SEGMENT_TYPE Ethernet (* Ethernet Segment *)
  (* Standard: 61499 ITA; Description: Copyright (c) 2008 Profactor GmbH This program and the accompanying materials are made available under the terms of the Eclipse Public License 2.0 which is available at https://www.eclipse.org/legal/epl-2.0/ SPDX-License-Identifier: EPL-2.0 *)
  (* Version 0.1, 2008-06-02, Gerhard Ebenhofer, Profactor GmbH, Initial version *)
  (* Version 3.0, 2025-04-14, Patrick Aigner, changed package *)
  PACKAGE iec61499::system;
END_SEGMENT_TYPE
